// TIA Portal V15.1 export
// export: Created 2024-05-17T05:38:05.7839536Z, ExportSetting WithDefaults, DisplayName Totally Integrated Automation Portal, DisplayVersion V15.1 Update 5, DisplayName TIA Portal Openness, DisplayVersion V15.1 Update 5, DisplayName SINAMICS Startdrive Advanced, DisplayVersion V15.1, DisplayName G130, G150, S120, S150, SINAMICS MV, S210, DisplayVersion V15.1, DisplayName G110M, G120, G120C, G120D, G120P, DisplayVersion V15.1, DisplayName STEP 7 Professional, DisplayVersion V15.1 Update 5, DisplayName STEP 7 Safety, DisplayVersion V15.1, DisplayName WinCC Professional, DisplayVersion V15.1 Update 5, DisplayName SIMATIC Visualization Architect, DisplayVersion V15.1
ORGANIZATION_BLOCK "I/O_FLT2"   // OB83, FBD, PullOrPlugOfModules
TITLE = "I/O Point Fault"
{ S7_Optimized_Access := 'TRUE' }
AUTHOR : VCC
VERSION : 0.0.0.0
// =============================================================================
// I/O Point Fault
// =============================================================================
// stored: IsIECCheckEnabled true, SetENOAutomatically False
   VAR_INPUT
      LADDR : HW_IO;   // Hardware identifier
      Event_Class : Byte;   // 16#38/39: module inserted, removed
      Fault_ID : Byte;   // Fault identifier
   END_VAR
BEGIN

REGION Network 1: **** 1 - Inputs **** Incrementation of number of executions
   // Incrementation of number of executions
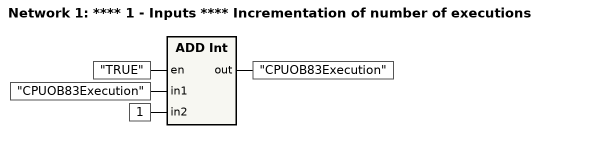
   IF "TRUE" THEN "CPUOB83Execution" := "CPUOB83Execution" + 1; END_IF;
END_REGION
END_ORGANIZATION_BLOCK
